Fanuc KAREL source: kt00048.KL

-- PROVISIONAL review KL for V940-1; original PC SHA256 4c4daf22f05507608e7486649c9b1c79760d049fad5c99adfd4f905f576c47f5
-- Incomplete behavior may be omitted. Consult companion uncertainty JSON. Do not deploy.
PROGRAM KT00048
%NOLOCKGROUP
VAR
  R1 : REAL
  OUT : REAL
-- UNRESOLVED_DECL H2 type=002017
BEGIN
  -- V9_ZERO_TABLE_METADATA_HINT layout=0001; no indexed target words; source/name/runtime held
  -- UNRESOLVED_PC offsets 5-16; opcodes 2E,23
  -- UNRESOLVED_PC offsets 21-35; opcodes 2E,22,9D,33,B4
  -- UNRESOLVED_PC offsets 40-63; opcodes 21,22,9D,33,B3,64,6A,23
  -- UNRESOLVED_PC offsets 68-72; opcodes 7F
END KT00048
